INTERFACE IDictionary EXTENDS IReadOnlyDictionary

METHOD Clear
END_METHOD

METHOD RemoveAt
VAR_INPUT
	index : DINT;
END_VAR
END_METHOD

METHOD Set : DINT
VAR_INPUT
	key : ANY;
	value : ANY;
	valueIsObject : BOOL := FALSE;
END_VAR
END_METHOD

METHOD SetGeneric : DINT
VAR_INPUT
	key : GENERIC_VALUE;
	value : GENERIC_VALUE;
END_VAR
END_METHOD

METHOD TryRemove : BOOL
VAR_INPUT
	key : ANY;
END_VAR
END_METHOD

END_INTERFACE

(* stored: Version 1.1.0.1
   Itf IDictionary: Id {57e81792-3900-4cad-861e-9c1a745a287a}
   Method Clear: Id {b1563b71-bd6a-4263-830c-984583112e42}
   Method RemoveAt: Id {a1586ec5-b74e-4671-96ad-ae4197067882}
   Method Set: Id {f13fbbaa-2923-411c-9a7c-638998bcf36d}
   Method SetGeneric: Id {9a515aa5-db44-4d5d-9fbd-7695318ffa56}
   Method TryRemove: Id {2539d3ce-1d3f-4331-818e-1181097b6910} *)
